Staubli VAL3: itemList.pgx

program itemList(string& x_sEvent[])
  local num l_nSize
  local string l_sEvent
  local num l_nKey
  local num i
  local string l_sMessage
  local string l_sPath
  local num l_nResult
  local string l_sToto
begin
  //
  // USE this procedure to view the items
  // list that you have already save
  //
  cls()
  //
  if x_sEvent=="PROG"
    // Prog
    l_sPath="Disk://instruction/PROG"
  else
    // other
    l_sPath=x_sEvent
    call getPath(l_sPath)
  endIf
  // reload the instruction
  l_nResult=instruction:libLoad(l_sPath)
  delay(0)
  //
  if l_nResult==0
    //
    call instruction:onInsert(x_sEvent)
  else
    popUpMsg("error loading "+x_sEvent+" "+l_sPath+" "+toString("",l_nResult))
  endIf
end
